FUNCTION_BLOCK NodeFinder_HMI (* Service Interface Function Block Type *)
  (* Standard: 61499-2 *)
  (* Version 0.0, 2/5/2024, midxav, template *)
  PACKAGE Main;
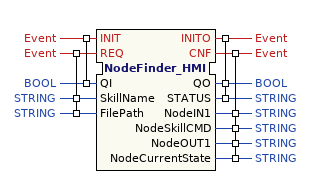
  EVENT_INPUT
    INIT WITH QI;
    REQ WITH SkillName, FilePath;
  END_EVENT
  EVENT_OUTPUT
    INITO WITH QO, STATUS;
    CNF WITH NodeIN1, NodeSkillCMD, NodeOUT1, NodeCurrentState;
  END_EVENT
  VAR_INPUT
    QI : BOOL;
    SkillName : STRING;
    FilePath : STRING;
  END_VAR
  VAR_OUTPUT
    QO : BOOL; (* Event Output Qualifier *)
    STATUS : STRING; (* Service Status *)
    NodeIN1 : STRING;
    NodeSkillCMD : STRING;
    NodeOUT1 : STRING;
    NodeCurrentState : STRING;
  END_VAR
  SERVICE /
    SEQUENCE 
    END_SEQUENCE
  END_SERVICE
END_FUNCTION_BLOCK
